// TIA Portal V19 export
FUNCTION "DEBUG_Simulate_Send_Msg_101" : Void   // FC216, LAD
TITLE = TEST INVIO MESSAGGIO 101
// stored: SetENOAutomatically false
   VAR_TEMP   // added for the SCL form of the ladder/FBD networks
      _w1 : Bool;
   END_VAR
BEGIN

REGION Network 1
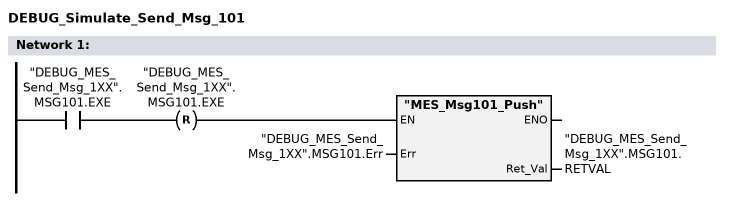
   RUNG wire#powerrail
      Contact( "DEBUG_MES_Send_Msg_1XX".MSG101.EXE )
      R_Coil( "DEBUG_MES_Send_Msg_1XX".MSG101.EXE )
      "MES_Msg101_Push"(Err := "DEBUG_MES_Send_Msg_1XX".MSG101.Err, Ret_Val => "DEBUG_MES_Send_Msg_1XX".MSG101.RETVAL)
   END_RUNG
   // the same network as SCL:
   #_w1 := "DEBUG_MES_Send_Msg_1XX".MSG101.EXE;
   IF #_w1 THEN
       "DEBUG_MES_Send_Msg_1XX".MSG101.EXE := FALSE;
       "DEBUG_MES_Send_Msg_1XX".MSG101.RETVAL := "MES_Msg101_Push"(Err := "DEBUG_MES_Send_Msg_1XX".MSG101.Err);
   END_IF;
END_REGION
END_FUNCTION
